(* PLC project Unnamed, Unknown Unnamed 1 *)
(* stored: creationDateTime 2022-06-03T13:37:24, modificationDateTime 2024-02-23T11:13:18 *)

PROGRAM blank_project
  VAR
    dummy_in AT %IX0.0 : BOOL;
    dummy_out AT %QX0.1 : BOOL;
  END_VAR

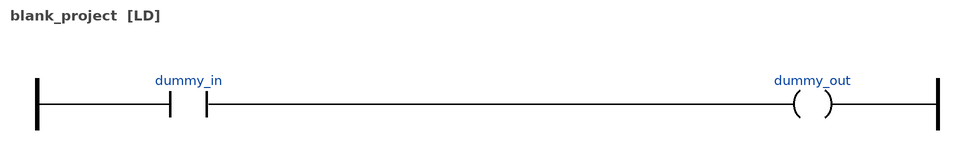
(* LD diagram, written out as Structured Text *)
dummy_out := dummy_in;
END_PROGRAM

CONFIGURATION Config0
  RESOURCE Res0 ON PLC
    TASK task0(INTERVAL := T#20ms, PRIORITY := 0);
    PROGRAM instance0 WITH task0 : blank_project;
  END_RESOURCE
END_CONFIGURATION
